Fanuc KAREL source: kt00294.KL

-- PROVISIONAL review KL for V940-1; original PC SHA256 bb7df9a6295899873218d9bf80e927b9e921f23aa938d8e4a67d5555240ee23f
-- Incomplete behavior may be omitted. Consult companion uncertainty JSON. Do not deploy.
PROGRAM KT00294
%NOLOCKGROUP
VAR
  I1 : INTEGER
  R2 : REAL
  OUT : BOOLEAN
BEGIN
  -- V9_ZERO_TABLE_METADATA_HINT layout=0001; no indexed target words; source/name/runtime held
  -- UNRESOLVED_PC offsets 5-16; opcodes 2E,23
  -- UNRESOLVED_PC offsets 21-32; opcodes 2E,23
  -- UNRESOLVED_PC offsets 37-58; opcodes 21,21,29,64,6E,23
  -- UNRESOLVED_PC offsets 63-67; opcodes 7F
END KT00294
